Staubli VAL3: printNum2d.pgx

public program printNum2d(num& x_nInput[] (dimensions=2))
  local num l_nElement
  local num l_nLength
  local num l_nRow
  local num l_RowResult
  local string l_sRow
begin

  for l_nRow = 0 to size(x_nInput,1)-1
    call extractRow(x_nInput, l_nRow, nRowResult)
    l_sRow = ""
    for l_nElement = 0 to size(nRowResult)-1
      l_sRow = l_sRow + toString(".3", nRowResult[l_nElement])
    endFor
    ? l_sRow
    endFor

end
